// TIA Portal V20 export
TYPE "typeReceipe"
// stored: Access Published, Namespace Unit1
   STRUCT
      processUnitNo : Int;
      selectedRecipeTypeID : Int;
      selectedRecipeID : Int;
      currentRecipeName : WString;
      currentRecipeID : Int;
   END_STRUCT;
END_TYPE
